// SIMATIC S7-200 SMART project (STEP 7-Micro/WIN SMART), CPU ST40

SYMBOL_TABLE System Symbols
Always_On        SM0.0    // Always ON
First_Scan_On    SM0.1    // ON for the first scan cycle only
END_SYMBOL_TABLE

ORGANIZATION_BLOCK Program_Block:OB1
TITLE=Program Comments
BEGIN
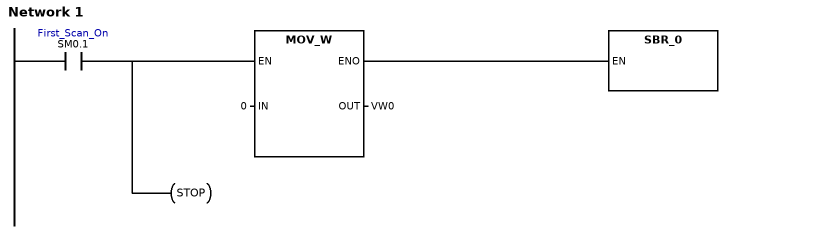
Network 1
LD     First_Scan_On:SM0.1
LPS
MOVW   0, VW0
AENO
CALL   SBR_0:SBR0
LPP
STOP
END_ORGANIZATION_BLOCK

SUBROUTINE_BLOCK SBR_0:SBR0
TITLE=Subroutine Comments
BEGIN
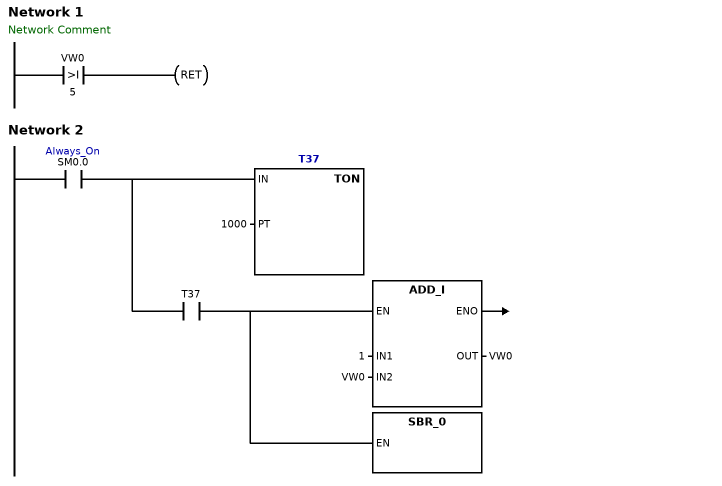
Network 1
// Network Comment
LDW>   VW0, 5
CRET
Network 2
LD     Always_On:SM0.0
TON    T37, 1000
A      T37
+I     1, VW0
CALL   SBR_0:SBR0
END_SUBROUTINE_BLOCK
